(*This function block does basic controls for the Ebara EV-A  pump. Turns off pump
in the event of errors/ warnings. Provides interlocking interface.*)
FUNCTION_BLOCK FB_EbaraEVA
VAR_INPUT
	i_xExtIlkOK	:	BOOL;
END_VAR
VAR_OUTPUT
	{attribute 'pytmc' := '
    pv: 
	'}
	stPump	:	ST_EbaraEVA; //Ebara dry pump structure 
END_VAR
VAR
	(*IO*)
	q_xRunDo AT%Q* : BOOL; // Output signal
	q_xRemote At%Q* :BOOL;// Remote/Local Control
	i_xAlarmOK AT%I* :BOOL; // Normally closed Alarm bit
	i_xIsRun   AT%I*:BOOL; // Input status
END_VAR


stPump.xIlkOK := i_xExtIlkOK AND stPump.i_xAlarmOK ;

IF stPump.xIlkOK THEN

	stPump.q_xRunDO := stPump.pv_xRunSW;
	ELSE
		stPump.PV_xRunSW := FALSE;
        stPump.q_xRunDO := FALSE;	
END_IF
//IO Mapping
ACT_IO();

ACTION ACT_IO:
stPump.i_xAlarmOK:=	i_xAlarmOK;
stPump.xErr := NOT(i_xAlarmOK);
stPump.i_xIsRun := i_xIsRun;
(*outputs*)
q_xRunDo:=stPump.q_xRunDo;
q_xRemote:= stPump.q_xRemote;
END_ACTION

END_FUNCTION_BLOCK

(* stored: Version 1.1.0.1, ProductVersion 3.1.4022.12
   POU FB_EbaraEVA: Id {fcf97f55-51a9-4ad7-88f0-a45e9e26409c}, SpecialFunc None
   Action ACT_IO: Id {1807940c-3fbb-4008-9507-5845d2fff7d5} *)
